(* IEC 61131-3 sources: eCockpitGit/test_project/src/%F%00 Library/%F%Structured Buffer Read Write Base/%ITF%ITF_StructWriterBase/%F%Structure, 3 files *)

(* ---- %METH%addKey.st ---- *)
//This method adds a key of any size to the current stuct/object
//It only works within structs/objects
METHOD addKey : BOOL
VAR_INPUT
	name			:POINTER TO EASCII;	//Address of string for the tag name text
END_VAR

(*%!%__DELIMITER__%!%*)

(* ---- %METH%arrayStart.st ---- *)
//This method starts an object or array
METHOD arrayStart : BOOL;
VAR_INPUT
	singleLine		:BOOL;
END_VAR
(*%!%__DELIMITER__%!%*)

(* ---- %METH%objectStart.st ---- *)
//This method starts an object or array
METHOD objectStart : BOOL;
VAR_INPUT
	singleLine		:BOOL;
END_VAR
(*%!%__DELIMITER__%!%*)
